INTERFACE ITcoMessages

(*~
		<docu>
			<summary>
				Adds message of 'debug' category to the message queue.				 
			</summary>		
		</docu>
~*)
METHOD PUBLIC Debug : ITcoMessageProperties
VAR_INPUT
	(*~
		<docu>
			<summary>
				Arbitrary message string.			 
			</summary>			
		</docu>
	~*)
	Message : STRING(TcoMessengerSettings.MAX_MESSAGE_TEXT_LENGHT);
END_VAR
END_METHOD

(*~
		<docu>
			<summary>
				Adds message of 'error' category to the message queue.				 
			</summary>						
		</docu>
~*)
METHOD PUBLIC Error : ITcoMessageProperties
VAR_INPUT
	(*~
		<docu>
			<summary>
				Arbitrary message string.			 
			</summary>			
		</docu>
	~*)
	Message : STRING(TcoMessengerSettings.MAX_MESSAGE_TEXT_LENGHT);
END_VAR
END_METHOD

(*~
		<docu>
			<summary>
				Adds message of 'information' category to the message queue.				 
			</summary>			
		</docu>
~*)
METHOD PUBLIC Info : ITcoMessageProperties
VAR_INPUT
	(*~
		<docu>
			<summary>
				Arbitrary message string.			 
			</summary>			
		</docu>
	~*)
	Message : STRING(TcoMessengerSettings.MAX_MESSAGE_TEXT_LENGHT);
END_VAR
END_METHOD

(*~
		<docu>
			<summary>
				Adds message of 'notification' category to the message queue.				 
			</summary>				
		</docu>
~*)
METHOD Notify  : ITcoMessageProperties
VAR_INPUT
	(*~
		<docu>
			<summary>
				Arbitrary message string.			 
			</summary>			
		</docu>
	~*)
	Message : STRING(TcoMessengerSettings.MAX_MESSAGE_TEXT_LENGHT);
END_VAR
END_METHOD

(*~
		<docu>
			<summary>
				Adds message of given category to the message queue.				 
			</summary>	
			<returns>Message index.</returns>		
		</docu>
~*)
METHOD PUBLIC Post  : ITcoMessageProperties
VAR_INPUT
	(*~
		<docu>
			<summary>
				Arbitrary message string.			 
			</summary>			
		</docu>
	~*)
	Message : STRING(TcoMessengerSettings.MAX_MESSAGE_TEXT_LENGHT);
	(*~
		<docu>
			<summary>
				Message category.			 
			</summary>			
		</docu>
	~*)
	Category : eMessageCategory;	
END_VAR
END_METHOD

(*~
		<docu>
			<summary>
				Adds message of 'programming error' category to the message queue.				 
			</summary>				
		</docu>
~*)
METHOD PUBLIC Programming : ITcoMessageProperties
VAR_INPUT
	(*~
		<docu>
			<summary>
				Arbitrary message string.			 
			</summary>			
		</docu>
	~*)
	Message : STRING(TcoMessengerSettings.MAX_MESSAGE_TEXT_LENGHT);
END_VAR
END_METHOD

(*~
		<docu>
			<summary>
				Adds message of 'trace' category to the message queue.				 
			</summary>					
		</docu>
~*)
METHOD PUBLIC Trace : ITcoMessageProperties
VAR_INPUT
	(*~
		<docu>
			<summary>
				Arbitrary message string.			 
			</summary>			
		</docu>
	~*)
	Message : STRING(TcoMessengerSettings.MAX_MESSAGE_TEXT_LENGHT);
END_VAR
END_METHOD

(*
	<docu>
		<summary>
			Unpins this messenger.
		</summary>
	</docu>
*) 
METHOD UnPin
END_METHOD

(*~
		<docu>
			<summary>
				Adds message of 'warning' category to the message queue.				 
			</summary>					
		</docu>
~*)
METHOD PUBLIC Warning : ITcoMessageProperties
VAR_INPUT
	(*~
		<docu>
			<summary>
				Arbitrary message string.			 
			</summary>			
		</docu>
	~*)
	Message : STRING(TcoMessengerSettings.MAX_MESSAGE_TEXT_LENGHT);
END_VAR
END_METHOD

END_INTERFACE

(* stored: Version 1.1.0.1
   Itf ITcoMessages: Id {5c5e06c8-fdc3-0a80-1edb-cded22f3b41d}
   Method Debug: Id {018dddc2-e993-08f8-07d7-a1616590828e}
   Method Error: Id {8a9b7711-5507-0817-347a-7f9d168058de}
   Method Info: Id {2900bcfb-ef3e-0cf3-1447-2675bc64b38e}
   Method Notify: Id {f3eeec7e-3765-03b9-22ed-50c217ca3deb}
   Method Post: Id {d3ce87bb-ac32-0271-2ca0-fcd31081c921}
   Method Programming: Id {de40152f-2593-0baa-37b5-73116b62afc0}
   Method Trace: Id {a2259cc4-50f1-0828-31e5-8e38d344d814}
   Method UnPin: Id {fabdeea1-c654-0144-0a58-11c0e4dd49f9}
   Method Warning: Id {ed68fc65-6b23-0ebe-2833-4b29338b28ec} *)
